{attribute 'qualified_only'}
VAR_GLOBAL CONSTANT
	EL3064MaxValueH	: REAL := 16383; //0~5V Half Input
	EL3064MaxValue 	: REAL := 32767; //0~10V
	EL4004MaxValueH	: REAL := 16383; //0~5V Half Output
	EL4004MaxValue 	: REAL := 32767; //4~20mA
	
	NumAnalogController :UINT:=29;
	nNumController	: INT := 18 ; //MFC 12EA, EPC 4ea
	nNumMFC			: INT := 12;
END_VAR

(* stored: Version 1.1.0.1, ProductVersion 3.1.4024.15
   GVL GVL_CONSTANT: Id {98785915-f5a2-4621-8795-7e3f35033e2f} *)
